(* B4 = Suspend Movement *)
TYPE ST_B4Res :
STRUCT
	PathID			:UINT;		(* 2 bytes*)
	CRC1			:BYTE;	    (* 1 byte*)
	CRC2			:BYTE;	    (* 1 byte*)		
	
END_STRUCT
END_TYPE

(* stored: Version 1.1.0.1, ProductVersion 3.1.4020.12
   DUT ST_B4Res: Id {fc34826c-84e5-4bd9-9551-8eb306f2efd3} *)
